// Core §3.8a — one client-defined named model field
TYPE ST_ModelField : STRUCT  Name : STRING(32);  Value : STRING(64);  END_STRUCT END_TYPE

(* stored: Version 1.1.0.1, ProductVersion 3.1.4024.12
   DUT ST_ModelField: Id {a1c7be5c-9477-42ca-b899-bfddb5108f64} *)
